Fanuc KAREL source: sys_pns2sr.kl

PROGRAM sys_pns2sr
%NOBUSYLAMP
%NOLOCKGROUP

VAR
	out_reg : INTEGER
%from tpe.klh %import get_int_arg
%from registers.klh %import set_string
%from systemlib.klh %import pns_to_str

BEGIN
	out_reg = tpe__get_int_arg(1)
	registers__set_string(out_reg, system__pns_to_str)
END sys_pns2sr
